FUNCTION_BLOCK FB_Mode
VAR_INPUT
	Men:BOOL;
	Material:BOOL;
	Rock:BOOL;
	Manual_switch:BOOL;
	Auto_switch:BOOL;
	Rope_capping_switch:BOOL;
	Brake_maint_switch:BOOL;
	Single_lever_control:BOOL;
END_VAR
VAR_OUTPUT
	cs_Mode_change:BOOL;
	cs_Men_rock_sw_fault:BOOL;
	cs_Auto_manual_sw_fault:BOOL;
	cs_Men_to_rock:BOOL;
	cs_Rock_to_men:BOOL;
	cs_Auto_to_manual:BOOL;
	cs_Manual_to_auto:BOOL;
	cs_Rope_capping_on:BOOL;
	cs_Rope_capping_off:BOOL;
	cs_Brake_maint_on:BOOL;
	cs_Brake_maint_off:BOOL;
	hmi_Status:WORD;
END_VAR
VAR
	F_TRIG_0: F_TRIG;
	R_TRIG_0: R_TRIG;
	R_TRIG_1: R_TRIG;
	F_TRIG_1: F_TRIG;
	R_TRIG_2: R_TRIG;
	F_TRIG_2: F_TRIG;
	R_TRIG_3: R_TRIG;
	F_TRIG_3: F_TRIG;
	R_TRIG_4: R_TRIG;
	F_TRIG_4: F_TRIG;
	R_TRIG_5: R_TRIG;
	F_TRIG_5: F_TRIG;
	TON_0: TON;
	BIT_TO_WORD_V0_0: FB_BIT_TO_WORD_V0;
END_VAR

Mode();
Mode_faults();

METHOD Mode
VAR_INPUT
END_VAR

VAR
END_VAR
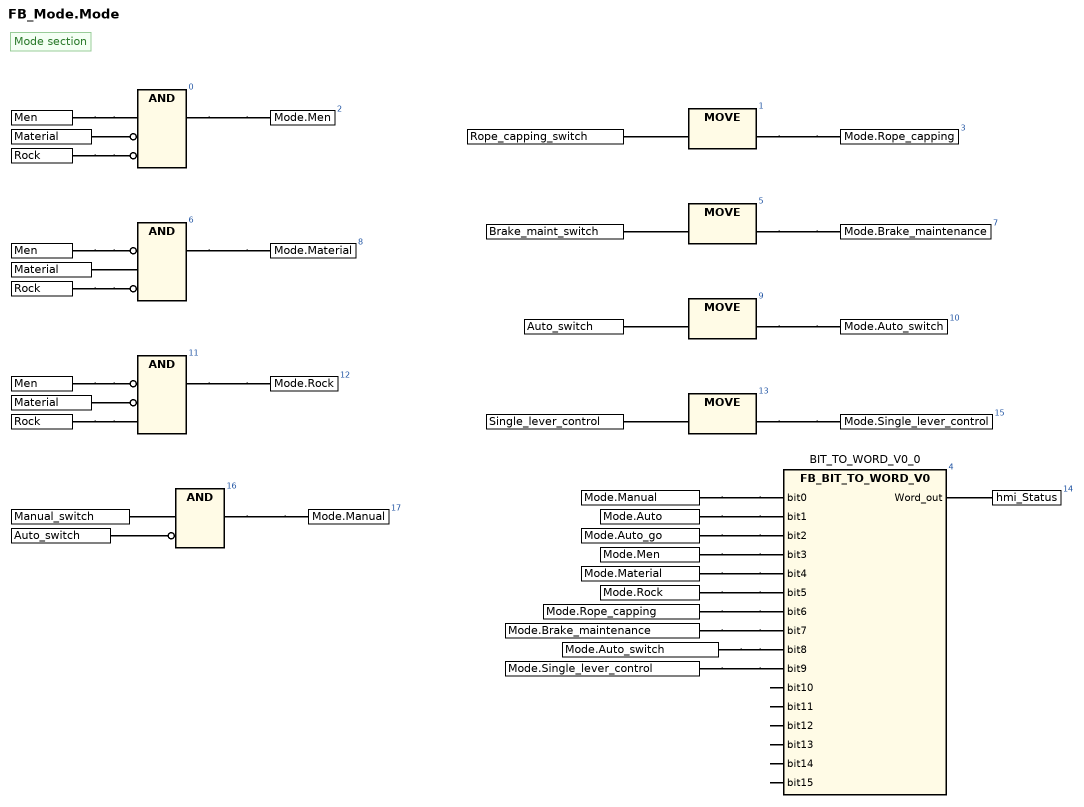
// Mode section
Mode.Men := Men AND NOT Material AND NOT Rock;
Mode.Rope_capping := Rope_capping_switch;
BIT_TO_WORD_V0_0(
    bit0 := Mode.Manual,
    bit1 := Mode.Auto,
    bit2 := Mode.Auto_go,
    bit3 := Mode.Men,
    bit4 := Mode.Material,
    bit5 := Mode.Rock,
    bit6 := Mode.Rope_capping,
    bit7 := Mode.Brake_maintenance,
    bit8 := Mode.Auto_switch,
    bit9 := Mode.Single_lever_control); // FB_BIT_TO_WORD_V0
Mode.Brake_maintenance := Brake_maint_switch;
Mode.Material := NOT Men AND Material AND NOT Rock;
Mode.Auto_switch := Auto_switch;
Mode.Rock := NOT Men AND NOT Material AND Rock;
hmi_Status := BIT_TO_WORD_V0_0.Word_out;
Mode.Single_lever_control := Single_lever_control;
Mode.Manual := Manual_switch AND NOT Auto_switch;
END_METHOD

METHOD Mode_faults
VAR_INPUT
END_VAR
VAR_INST // added by the converter: edge detectors and wires of the graphical bodies
    _w1, _w2, _w3 : BOOL;
END_VAR
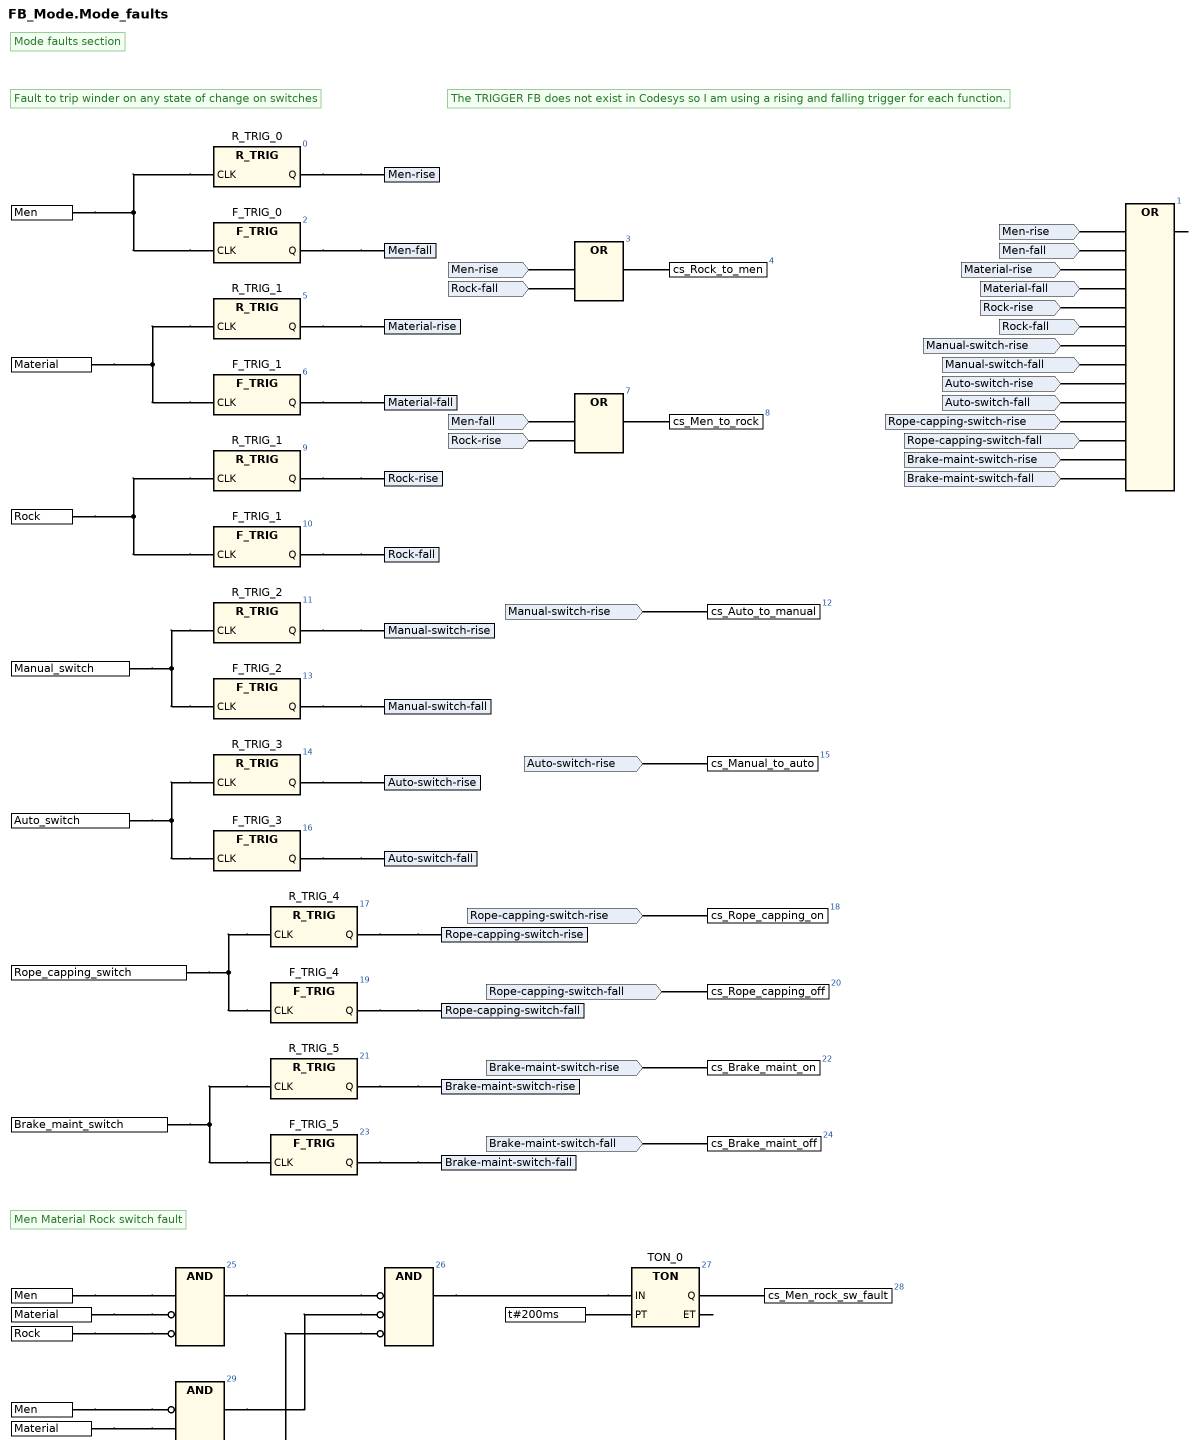
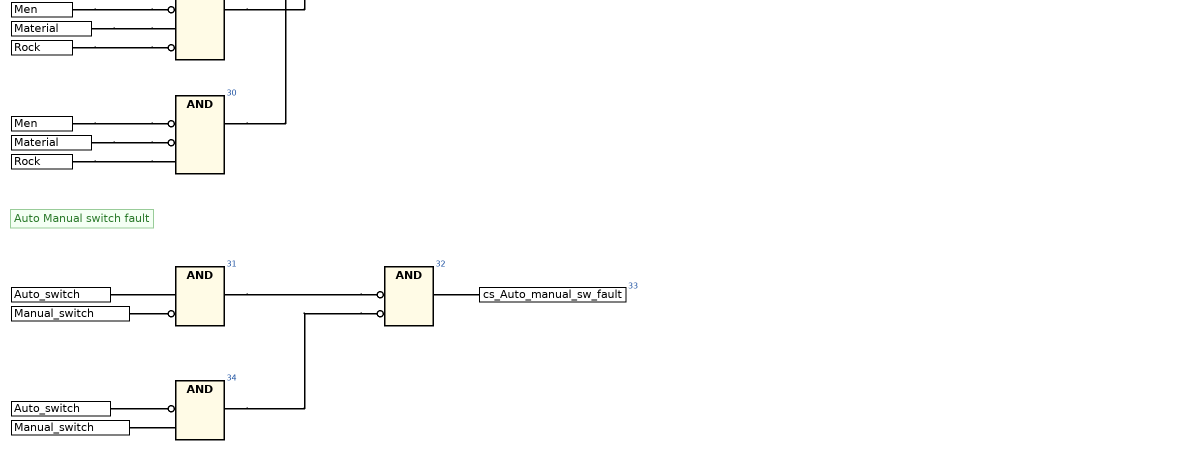
// Mode faults section
// Fault to trip winder on any state of change on switches
// The TRIGGER FB does not exist in Codesys so I am using a rising and falling trigger for each function.
R_TRIG_0(CLK := Men); // R_TRIG
(* R_TRIG_0.Q OR F_TRIG_0.Q OR R_TRIG_1.Q OR F_TRIG_1.Q OR R_TRIG_1.Q OR F_TRIG_1.Q OR R_TRIG_2.Q OR F_TRIG_2.Q OR R_TRIG_3.Q OR F_TRIG_3.Q OR R_TRIG_4.Q OR F_TRIG_4.Q OR R_TRIG_5.Q OR F_TRIG_5.Q; result not used *)
F_TRIG_0(CLK := Men); // F_TRIG
cs_Rock_to_men := R_TRIG_0.Q OR F_TRIG_1.Q;
R_TRIG_1(CLK := Material); // R_TRIG
F_TRIG_1(CLK := Material); // F_TRIG
cs_Men_to_rock := F_TRIG_0.Q OR R_TRIG_1.Q;
R_TRIG_1(CLK := Rock); // R_TRIG
F_TRIG_1(CLK := Rock); // F_TRIG
R_TRIG_2(CLK := Manual_switch); // R_TRIG
cs_Auto_to_manual := R_TRIG_2.Q;
F_TRIG_2(CLK := Manual_switch); // F_TRIG
R_TRIG_3(CLK := Auto_switch); // R_TRIG
cs_Manual_to_auto := R_TRIG_3.Q;
F_TRIG_3(CLK := Auto_switch); // F_TRIG
R_TRIG_4(CLK := Rope_capping_switch); // R_TRIG
cs_Rope_capping_on := R_TRIG_4.Q;
F_TRIG_4(CLK := Rope_capping_switch); // F_TRIG
cs_Rope_capping_off := F_TRIG_4.Q;
R_TRIG_5(CLK := Brake_maint_switch); // R_TRIG
cs_Brake_maint_on := R_TRIG_5.Q;
F_TRIG_5(CLK := Brake_maint_switch); // F_TRIG
cs_Brake_maint_off := F_TRIG_5.Q;
// Men Material Rock switch fault
TON_0(IN := NOT (Men AND NOT Material AND NOT Rock) AND NOT _w1 AND NOT _w2, PT := t#200ms); // TON
cs_Men_rock_sw_fault := TON_0.Q;
_w1 := NOT Men AND Material AND NOT Rock;
_w2 := NOT Men AND NOT Material AND Rock;
// Auto Manual switch fault
cs_Auto_manual_sw_fault := NOT (Auto_switch AND NOT Manual_switch) AND NOT _w3;
_w3 := NOT Auto_switch AND Manual_switch;
END_METHOD

END_FUNCTION_BLOCK

(* stored: Version 1.1.0.1, ProductVersion 3.1.4024.0
   POU FB_Mode: Id {b9c44bc0-8485-40f2-ab8f-779455cede2d}, SpecialFunc None
   Method Mode: Id {9776f3e0-0065-41d3-a038-eb6103234711}
   Method Mode_faults: Id {fa5ce039-80cd-4b4e-96dd-1d52d703c3a9} *)
